# EPICS autosave request: caenN1470/caenN1470chan_settings.req
$(P)$(Q):ISET$(CHAN)
$(P)$(Q):ON$(CHAN)
$(P)$(Q):RDW$(CHAN)
$(P)$(Q):RUP$(CHAN)
$(P)$(Q):UPDATE$(CHAN).SCAN
$(P)$(Q):VSET$(CHAN)
